FUNCTION_BLOCK Controller
  (* Standard: 61499-2 *)
  (* Version 0,1, 2015-00-14, Th?o, PC_THEO *)
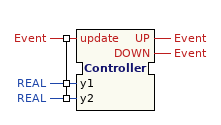
  EVENT_INPUT
    update WITH y1, y2;
  END_EVENT
  EVENT_OUTPUT
    UP;
    DOWN;
  END_EVENT
  VAR_INPUT
    y1 : REAL;
    y2 : REAL;
  END_VAR
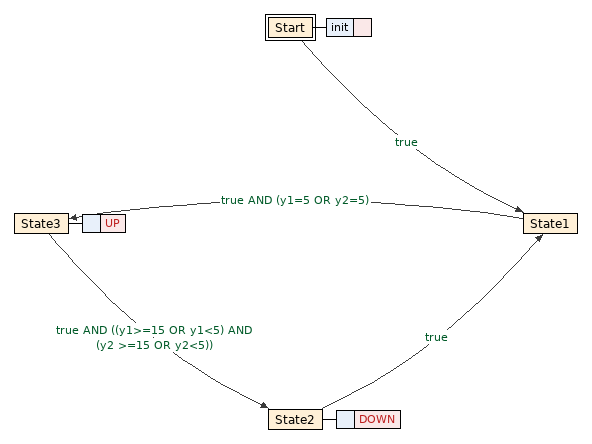
  EC_STATES
    Start : init;
    State1;
    State2 : -> DOWN;
    State3 : -> UP;
  END_STATES
  EC_TRANSITIONS
    Start TO State1 := true;
    State1 TO State3 := true AND (y1=5 OR y2=5);
    State2 TO State1 := true;
    State3 TO State2 := true AND ((y1>=15 OR y1<5) AND (y2 >=15 OR y2<5));
  END_TRANSITIONS
  ALGORITHM init IN C:
me->y1=0;
me->y2=0;
  END_ALGORITHM
END_FUNCTION_BLOCK
